// File: DB_ScadaToPlc_ManualMechCmd.scl
DATA_BLOCK "DB_ScadaToPlc_ManualMechCmd"
{ S7_Optimized_Access := 'TRUE' }

VAR
    // по одному елементу на кожен слот DB_Mechs.Mechs[0..255]
    CmdBySlot : ARRAY[0..255] OF "UDT_ManualMechCmdItem";
END_VAR

BEGIN
END_DATA_BLOCK
